// TIA Portal V18 export
// export: Created 2026-01-09T11:23:28.7100827Z, ExportSetting WithDefaults, DisplayName Totally Integrated Automation Portal, DisplayVersion V18 Update 5, DisplayName TIA Portal Openness, DisplayVersion V18 Update 5, DisplayName TIA Portal Teamcenter Gateway, DisplayVersion V18, DisplayName TIA Portal Version Control Interface, DisplayVersion V18, DisplayName SINAMICS Startdrive Advanced, DisplayVersion V18 SP2 Update 1, DisplayName SINAMICS Startdrive G110M, G120, G120C, G120D, G120P, G115D, DisplayVersion V18 SP2 Update 1, DisplayName SINAMICS Startdrive G130, G150, S120, S150, SINAMICS MV, S210, G220, S200, DisplayVersion V18 SP2 Update 1, DisplayName STEP 7 Professional, DisplayVersion V18 Update 5, DisplayName STEP 7 Safety, DisplayVersion V18, DisplayName WinCC Professional, DisplayVersion V18 Update 5
Screen "200 ManualStructure"  1280x800, Number=198, Template=T1
  ScreenLayer "Layer_0"
    Button "btnMenu3" at 128,725 size 128x75  Mode=Text, StyleItem=BtnActive20, TextOff="手动 / Manual / Manuálny"
    Button "btnMenu4" at 384,725 size 128x75  Mode=Text, StyleItem=BtnNormal20
    Button "btnMenu5" at 512,725 size 128x75  Mode=Text, StyleItem=BtnNormal20
    Button "btnMenu6" at 640,725 size 128x75  Mode=Text, StyleItem=BtnNormal20
    Button "btnMenu7" at 896,725 size 128x75  Mode=Text, StyleItem=BtnNormal20
    Button "btnMenu8" at 1152,725 size 128x75  Mode=Graphic, PictureOff=图形_30, StyleItem=BtnNormal20
      on Press: ActivateScreen(Screen name := , Object number := 0); SetTag(Tag := Sys_VersionManagement_HMIPageID, Value := 220)
    Button "按钮_2" at 1151,265 size 128x75  Mode=Text, StyleItem=BtnNormal20
    Button "按钮_3" at 1151,435 size 128x75  Mode=Text, StyleItem=BtnNormal20
    Button "btnMenu8_1" at 1152,350 size 128x75  Mode=Text, StyleItem=BtnNormal20
    Button "按钮_4" at 0,265 size 128x75  Mode=Text, StyleItem=BtnNormal20, TextOff="C_涂胶 / C_Glue", TextOn="C_涂胶 / C_Glue"
      on Click: ActivateScreen(Screen name := 230_Cylinder, Object number := 0)
    Button "按钮_5" at 0,350 size 128x75  Mode=Text, StyleItem=BtnNormal20, TextOff="E_NG盒 / E_NG", TextOn="E_NG盒 / E_NG"
      on Click: ActivateScreen(Screen name := 240_Cylinder_E1, Object number := 0)
    Button "按钮_6" at 0,180 size 128x75  Mode=Text, StyleItem=BtnNormal20, TextOff="B_压机 / B_Press Kistler", TextOn="B_压机 / B_Press Kistler / B"
      on Click: ActivateScreen(Screen name := 220_Cylinder_B1, Object number := 0)
    Button "btnMenu8_3" at 0,435 size 128x75  Mode=Text, StyleItem=BtnNormal20, TextOff="F_机器人 / F_Robot", TextOn="F_机器人 / F_Robot"
      on Click: ActivateScreen(Screen name := 250_Cylinder_F1, Object number := 0)
    Button "btnMenu8_4" at 144,95 size 128x75  Mode=Text, StyleItem=BtnNormal20, TextOff="K_Reserve 上料//预留 / K_Reserve Loading", TextOn="K_Reserve 上料//预留 / K_Reserve Loading"
      on Click: ActivateScreen(Screen name := 280_Cylinder_K1, Object number := 0)
    Button "按钮_7" at 0,95 size 128x75  Mode=Text, StyleItem=BtnNormal20, TextOff="A_Ring上料 / A_RingTable", TextOn="A_Ring上料 / A_RingTable"
      on Click: ActivateScreen(Screen name := 210_Cylinder_A1, Object number := 0)
    Button "按钮_8" at 1151,95 size 128x75  Mode=Text, StyleItem=BtnNormal18, TextOff="安全门 / Safety Door / bezpečnostné dvere"
      on Press: ActivateScreen(Screen name := 201  SafetyGate, Object number := 0); SetTag(Tag := Sys_VersionManagement_HMIPageID, Value := 201)
    Button "btnMenu6_1" at 768,725 size 128x75  Mode=Text, StyleItem=BtnNormal20
    Button "btnMenu7_1" at 1024,725 size 128x75  Mode=Text, StyleItem=BtnNormal20
    Button "btnMenu8_5" at 0,520 size 128x75  Mode=Text, StyleItem=BtnNormal20, TextOff="H_Shaft 上料 / H_Shaft Loading", TextOn="H_Shaft 上料 / H_Shaft Loading"
      on Click: ActivateScreen(Screen name := 260_Cylinder_H1, Object number := 0)
    Button "按钮_9" at 1151,180 size 128x75  Mode=Text, PictureOff=向右箭头_0, StyleItem=BtnNormal20, TextOff="报 警 / Alarm"
      RangeAppearanceAnimation "RangeAppearanceAnimation"
        tag ST_AlarmON
        1..1: back #ff0000, fore #d6d3ce, flashing
      on Click: ActivateScreen(Screen name := 300Main, Object number := 0); SetTag(Tag := Sys_VersionManagement_HMIPageID, Value := 300)
    Button "按钮_10" at 1151,605 size 128x75  Mode=Text, PictureOff=向右箭头_0, StyleItem=BtnFunction20, TextOff="灯测试 / Test Lamp / Test svetel"
      RangeAppearanceAnimation "RangeAppearanceAnimation"
        tag ST_CommandTestLamp
        1..1: back #00ff00, fore #000000
      on Press: SetBit(Tag := ST_CommandTestLamp)
      on Release: ResetBit(Tag := ST_CommandTestLamp)
    GraphicView "图形视图_1" at 278,95 size 864x584  Picture=图形_44
    Button "btnMenu8_2" at 0,605 size 128x75  Mode=Text, StyleItem=BtnNormal20, TextOff="J_Magnet 上料 / J_Magnet Loading", TextOn="J_Magnet 上料 / J_Magnet Loading"
      on Click: ActivateScreen(Screen name := 270_Cylinder_J1, Object number := 0)
    Button "按钮_11" at 144,180 size 128x75  Mode=Text, StyleItem=BtnNormal20, TextOff="L_下料 / L_Unload", TextOn="L_下料 / L_Unload"
      on Click: ActivateScreen(Screen name := 290_Cylinder_L1, Object number := 0)
    Group "Group"
      Circle "圆_2" at 446,592 size 24x24
      Circle "圆_3" at 451,597 size 15x15
        RangeAppearanceAnimation "RangeAppearanceAnimation"
          tag HMI_ESTOP
          1..1: back #ff0000, fore #181c31, flashing
          0..0: back #ff0000, fore #181c31
    Group "Group_2"
      Circle "圆_6" at 314,473 size 24x24
      Circle "圆_7" at 319,478 size 15x15
        RangeAppearanceAnimation "RangeAppearanceAnimation"
          tag ESTOP_PB1
          1..1: back #ff0000, fore #181c31, flashing
          0..0: back #ff0000, fore #181c31
    Group "Group_3"
      Circle "圆_8" at 423,305 size 24x24
      Circle "圆_9" at 428,310 size 15x15
        RangeAppearanceAnimation "RangeAppearanceAnimation"
          tag ESTOP_PB7
          1..1: back #ff0000, fore #181c31, flashing
          0..0: back #ff0000, fore #181c31
    Group "Group_4"
      Circle "圆_10" at 384,122 size 24x24
      Circle "圆_11" at 389,127 size 15x15
        RangeAppearanceAnimation "RangeAppearanceAnimation"
          tag ESTOP_PB3
          1..1: back #ff0000, fore #181c31, flashing
          0..0: back #ff0000, fore #181c31
    Group "Group_5"
      Circle "圆_12" at 586,305 size 24x24
      Circle "圆_13" at 591,310 size 15x15
        RangeAppearanceAnimation "RangeAppearanceAnimation"
          tag ESTOP_PB8
          1..1: back #ff0000, fore #181c31, flashing
          0..0: back #ff0000, fore #181c31
    Group "Group_6"
      Circle "圆_14" at 734,305 size 24x24
      Circle "圆_15" at 739,310 size 15x15
        RangeAppearanceAnimation "RangeAppearanceAnimation"
          tag ESTOP_PB9
          1..1: back #ff0000, fore #181c31, flashing
          0..0: back #ff0000, fore #181c31
    Group "Group_7"
      Circle "圆_16" at 531,124 size 24x24
      Circle "圆_21" at 536,129 size 15x15
        RangeAppearanceAnimation "RangeAppearanceAnimation"
          tag ESTOP_PB4
          1..1: back #ff0000, fore #181c31, flashing
          0..0: back #ff0000, fore #181c31
    Group "Group_8"
      Circle "圆_22" at 677,124 size 24x24
      Circle "圆_23" at 682,129 size 15x15
        RangeAppearanceAnimation "RangeAppearanceAnimation"
          tag ESTOP_PB5
          1..1: back #ff0000, fore #181c31, flashing
          0..0: back #ff0000, fore #181c31
    Group "Group_9"
      Circle "圆_24" at 806,122 size 24x24
      Circle "圆_25" at 811,127 size 15x15
        RangeAppearanceAnimation "RangeAppearanceAnimation"
          tag ESTOP_PB6
          1..1: back #ff0000, fore #181c31, flashing
          0..0: back #ff0000, fore #181c31
    Group "Group_10"
      Circle "圆_26" at 1039,281 size 24x24
      Circle "圆_27" at 1044,286 size 15x15
        RangeAppearanceAnimation "RangeAppearanceAnimation"
          tag PilzData_85A1_I12
          0..0: back #ff0000, fore #181c31, flashing
          1..1: back #ff0000, fore #181c31
    Group "Group_12"
      Circle "圆_30" at 890,455 size 24x24
      Circle "圆_31" at 895,460 size 15x15
        RangeAppearanceAnimation "RangeAppearanceAnimation"
          tag ESTOP_PB2
          1..1: back #ff0000, fore #181c31, flashing
          0..0: back #ff0000, fore #181c31
    TextField "文本域_18" at 469,591 size 110x28  Text="HMI ESTOP"
    Group "Group_1"
      Circle "圆_4" at 1039,95 size 24x24
      Circle "圆_5" at 1044,100 size 15x15
        RangeAppearanceAnimation "RangeAppearanceAnimation"
          tag PilzData_85A1_I13
          0..0: back #ff0000, fore #181c31, flashing
          1..1: back #ff0000, fore #181c31
    TextField "Template_Text field_1" at 855,4 size 299x25  Text="MES在线 / Tool scanning code is running / MES online"
      RangeAppearanceAnimation "RangeAppearanceAnimation"
        tag ChangeOver_DB_Global_ScanFixtureFlag
        1..1: back #00ff00, fore #31344a, flashing
      SingleBitVisibilityAnimation "VisibilityAnimation"
        tag ChangeOver_DB_Global_ScanFixtureFlag
    Group "Group_11"
      Button "btnMenu7_2" at 306,520 size 107x46  Mode=Text, TextOff="A-Ring1 上料 / A-Load Ring1", TextOn="A-Ring1 上料 / A-Load Ring1"
        on Click: ActivateScreen(Screen name := 210_Cylinder_A1, Object number := 0)
      GraphicIOField "图形 I/O 域_9" at 306,520 size 36x46  Mode=InOutput, OnValue=1, PictureList=StationStatus
        ProcessValue := Status_A1TableScanStatus
    Group "Group_13"
      Button "btnMenu7_6" at 536,516 size 106x33  Mode=Text, TextOff="C-涂胶 / C-Glue", TextOn="C-涂胶 / C-Glue"
        on Click: ActivateScreen(Screen name := 230_Cylinder, Object number := 0)
      GraphicIOField "图形 I/O 域_15" at 536,516 size 36x33  Mode=InOutput, OnValue=1, PictureList=StationStatus
        ProcessValue := Status_C_Glue_Status
    Group "Group_14"
      Button "btnMenu7_5" at 795,520 size 108x46  Mode=Text, TextOff="A-Ring2 上料 / A-Load Ring2", TextOn="A-Ring2 上料 / A-Load Ring2"
        on Click: ActivateScreen(Screen name := 216_Cylinder_A2, Object number := 0)
      GraphicIOField "图形 I/O 域_14" at 795,520 size 36x46  Mode=InOutput, OnValue=1, PictureList=StationStatus
        ProcessValue := Status_A2TableScanStatus
    Group "Group_15"
      Button "btnMenu7_4" at 639,477 size 117x33  Mode=Text, TextOff="B-压机2 / B-Press2", TextOn="B-压机2 / B-Press2"
        on Click: ActivateScreen(Screen name := 227 Kistler_375A1, Object number := 0)
      GraphicIOField "图形 I/O 域_13" at 639,477 size 36x33  Mode=InOutput, OnValue=1, PictureList=StationStatus
        ProcessValue := Status_B2Press_Status
    Group "Group_16"
      Button "btnMenu7_12" at 323,170 size 105x64  Mode=Text, TextOff="H- 轴上料 / H- ShaftBelt", TextOn="H- 轴上料 / H- ShaftBelt"
        on Click: ActivateScreen(Screen name := 261_Motor_H1, Object number := 0); SetTag(Tag := Sys_VersionManagement_HMIPageID, Value := 261)
      GraphicIOField "图形 I/O 域_1" at 323,170 size 36x33  Mode=InOutput, OnValue=1, PictureList=StationStatus
        ProcessValue := StationStatusH
    Group "Group_17"
      Button "btnMenu7_16" at 484,170 size 105x64  Mode=Text, TextOff="J- 磁铁上料 / J- MagnetBelt", TextOn="J- 磁铁上料 / J- MagnetBelt"
        on Click: ActivateScreen(Screen name := 271_Motor_J1, Object number := 0); SetTag(Tag := Sys_VersionManagement_HMIPageID, Value := 271)
      GraphicIOField "图形 I/O 域_2" at 484,170 size 36x33  Mode=InOutput, OnValue=1, PictureList=StationStatus
        ProcessValue := StationStatusJ
    Group "Group_18"
      Button "btnMenu7_17" at 650,170 size 105x64  Mode=Text, TextOff="K-预留 上料//预留 / K- ReserveBelt", TextOn="K-预留 上料//预留 / K- ReserveBelt"
        on Click: ActivateScreen(Screen name := 281_Motor_K1, Object number := 0); SetTag(Tag := Sys_VersionManagement_HMIPageID, Value := 281)
      GraphicIOField "图形 I/O 域_3" at 650,170 size 36x33  Mode=InOutput, OnValue=1, PictureList=StationStatus
        ProcessValue := StationStatusK
    Group "Group_19"
      Button "btnMenu7_18" at 795,170 size 105x64  Mode=Text, TextOff="L- 空托盘 / L- UnloadBelt", TextOn="L- 空托盘 / L- UnloadBelt"
        on Click: ActivateScreen(Screen name := 291_Motor_L1, Object number := 0); SetTag(Tag := Sys_VersionManagement_HMIPageID, Value := 291)
      GraphicIOField "图形 I/O 域_4" at 795,170 size 36x33  Mode=InOutput, OnValue=1, PictureList=StationStatus
        ProcessValue := StationStatusL
    Group "Group_20"
      Button "btnMenu7_19" at 913,213 size 125x33  Mode=Text, TextOff="固化炉 / Solidify", TextOn="固化炉 / Solidify"
        on Click: ShowPopupScreen(Name of the screen := CuringOven, X coordinate := 350, Y coordinate := 150, Display mode := -1, Animation := -1, Animation speed := 1)
      GraphicIOField "图形 I/O 域_5" at 913,213 size 36x33  Mode=InOutput, OnValue=1, PictureList=StationStatus
        ProcessValue := Status_Solidify_Status
    Group "Group_21"
      Button "btnMenu7_20" at 350,362 size 120x33  Mode=Text, TextOff="F-机器人1 / F-Robot1", TextOn="F-机器人1 / F-Robot1"
        on Click: ActivateScreen(Screen name := 251  Robot_1, Object number := 0)
      GraphicIOField "图形 I/O 域_6" at 350,362 size 36x33  Mode=InOutput, OnValue=1, PictureList=StationStatus
        ProcessValue := Status_FRobot_1_Status
    Group "Group_22"
      Button "btnMenu7_21" at 566,362 size 120x33  Mode=Text, TextOff="F-机器人2 / F-Robot2", TextOn="F-机器人2 / F-Robot2"
        on Click: ActivateScreen(Screen name := 254  Robot_2, Object number := 0)
      GraphicIOField "图形 I/O 域_7" at 566,362 size 36x33  Mode=InOutput, OnValue=1, PictureList=StationStatus
        ProcessValue := Status_FRobot_2_Status
    Group "Group_23"
      Button "btnMenu7_22" at 716,362 size 120x33  Mode=Text, TextOff="F-机器人3 / F-Robot3", TextOn="F-机器人3 / F-Robot3"
        on Click: ActivateScreen(Screen name := 257  Robot_3, Object number := 0)
      GraphicIOField "图形 I/O 域_8" at 716,362 size 36x33  Mode=InOutput, OnValue=1, PictureList=StationStatus
        ProcessValue := Status_FRobot_3_Status
    Group "Group_24"
      Button "btnMenu7_24" at 281,417 size 138x38  Mode=Text, TextOff="E-NG盒1 / E-NG1", TextOn="E-NG盒1 / E-NG1"
        on Click: ActivateScreen(Screen name := 240_Cylinder_E1, Object number := 0)
      GraphicIOField "图形 I/O 域_11" at 281,417 size 47x38  Mode=InOutput, OnValue=1, PictureList=StationStatus
        ProcessValue := Status_ENG_1_Status
    Group "Group_25"
      Button "btnMenu7_3" at 389,477 size 119x33  Mode=Text, TextOff="B-压机1 / B-Press1", TextOn="B-压机1 / B-Press1"
        on Click: ActivateScreen(Screen name := 221 Kistler__372A1, Object number := 0)
      GraphicIOField "图形 I/O 域_12" at 389,477 size 36x33  Mode=InOutput, OnValue=1, PictureList=StationStatus
        ProcessValue := Status_B1Press_Status
    Group "Group_26"
      Button "btnMenu7_23" at 823,417 size 136x38  Mode=Text, TextOff="E-NG盒2 / E-NG2", TextOn="E-NG盒2 / E-NG2"
        on Click: ActivateScreen(Screen name := 246_Cylinder_E2, Object number := 0)
      GraphicIOField "图形 I/O 域_10" at 823,417 size 46x38  Mode=InOutput, OnValue=1, PictureList=StationStatus
        ProcessValue := Status_ENG_1_Status
    Button "btnMenu4_1" at 256,725 size 128x75  Mode=Text, StyleItem=BtnNormal20
    Button "按钮_1" at 1151,520 size 128x75  Mode=Text, StyleItem=BtnNormal20
